FUNCTION SECOND_OF_DT : INT
VAR_INPUT
	XDT : DT;
END_VAR


(*
	version 1.0	6. jun. 2008
	programmer 	oscat
	tested BY	oscat

SECOND_OF_DT returns the current second (second of minute) of a DT variable

*)

SECOND_OF_DT := DWORD_TO_INT(DT_TO_DWORD(XDT) MOD 60);

(* revision history
hm		6.9.2008	rev 1.0
	original version

*)

END_FUNCTION

(* stored: Version 1.1.0.1, ProductVersion 3.1.4022.7
   POU SECOND_OF_DT: Id {e217f2fc-8b57-4e3e-b681-162637405a98}, SpecialFunc None *)
